# EPICS substitutions: streamApp/pluginDb/pluginMagick.substitutions
#
# pluginMagick.substitutions
#

file NDFile.template
{
	{
    PORT            = "Magick\$(N)",
    P               = "$(CAM):",
	R				= "$(PORT):",
    ADDR            = "\$(ADDR=0)",
    TIMEOUT         = "\$(TIMEOUT=1)",
	}
}
file NDFileAutoFileNumber.template
{
	{
    PORT            = "Magick\$(N)",
    P               = "$(CAM):",
	R				= "$(PORT):",
	}
}
file NDFileMagick.template
{
	{
    PORT            = "Magick\$(N)",
    P               = "$(CAM):",
	R				= "$(PORT):",
    ADDR            = "\$(ADDR=0)",
    TIMEOUT         = "\$(TIMEOUT=1)",
    NDARRAY_PORT    = "\$(PLUGIN_SRC)",
    NDARRAY_ADDR    = "\$(NDARRAY_ADDR=0)",
	}
}
